{attribute 'qualified_only'}
VAR_GLOBAL
	fCyclicTime : LREAL := 0.01;
	bSimulationRunning : BOOL := FALSE;
END_VAR

(* stored: Version 1.1.0.1, ProductVersion 3.1.4024.10
   GVL Parameters: Id {3db240b4-cea9-499c-90bf-c853e658de87} *)
